PROGRAM POU
VAR
	
	i : INT := 0;
	f : REAL := 0.0;
	elapsed : TIME := TIME#0M0S0MS;
	today : DATE := DATE#2020-01-01;
	message : STRING := '';
	count : BYTE := 0;
	
	A AT %I* : BOOL := FALSE;
	B AT %I* : BOOL := FALSE;
	C AT %I* : BOOL := FALSE;
	D AT %Q* : BOOL := FALSE;
		
	op1 : INT := 1;
	op2 : INT := 2;
	res : REAL := 0.0;
	test : BOOL := FALSE;
	
	tmr1 : TON;
	
END_VAR

// Single line comment

(* 
	Multiple line comment
*)

// Structured Text statments

i := 0;
f := 0.0;
elapsed := T#1S;
today := D#2020-05-18;
message := 'Good Morning!';

// Operators (strongest to weakest binding)

res := MAX(op1,op2); // MAX() function

res := EXPT(op1, op2); // Exponentation operator

res := -op1; // Negation operator
B := NOT A; // NOT operator

res := op1 * op2; // * operator
res := op1 / op2; // / operator
res := op1 MOD op2; // MOD operator

res := op1 + op2; // + operator
res := op1 - op2; // - operator

test := op1 < op2; // < operator
test := op1 > op2; // > operator
test := op1 <= op2; // <= operator
test := op1 >= op2; // >= operator

test := op1 = op2; // = operator

C := A AND B; // AND operator

C := A XOR B; // XOR operator

C := A OR B; // OR operator

// IF statement

IF A = B THEN // IF statement
	D := TRUE;
END_IF

IF A = B THEN // IF-ELSE statement
	D := TRUE;
ELSE
	D := FALSE;
END_IF

IF A = B THEN // IF-ELSIF statement
	D := TRUE;
ELSIF A = C THEN
	D := FALSE;
END_IF

// CASE Statement

i := 0;

CASE i OF
	0: A := TRUE;
	1: B := TRUE;
	2: C := TRUE;
ELSE
	D := TRUE;
END_CASE

// FOR statement

f := 0.0;

FOR i := 0 TO 5 BY 1 DO // FOR loop
	f := f + i;
END_FOR

f := 0.0;

FOR i := 0 TO 5 BY 1 DO // FOR loop with EXIT statment
	f := f + i;
	
	IF f > 3 THEN
		EXIT;
	END_IF
END_FOR

// WHILE loop

i := 0;
f := 0.0;

WHILE f < 5 DO // WHILE loop
	f := f + i;
	i := i + 1;
END_WHILE

i := 0;
f := 0.0;

WHILE f < 5 DO // WHILE loop with EXIT statement
	f := f + i;
	i := i + 1;
	
	IF f > 3 THEN
		EXIT;
	END_IF
END_WHILE

// REPEAT loop

i := 0;
f := 0.0;

REPEAT // REPEAT loop
	f := f + i;
	i := i + 1;
UNTIL f >= 5
END_REPEAT

REPEAT // REPEAT loop with EXIT statment
	f := f + i;
	i := i + 1;
	
	IF f > 3 THEN
		EXIT;
	END_IF
UNTIL f = 5
END_REPEAT

// Timer

D := FALSE;
tmr1(IN := TRUE, PT := T#5S);

IF (tmr1.ET >= T#3S) THEN
	D := TRUE;
END_IF

END_PROGRAM

(* stored: Version 1.1.0.1, ProductVersion 3.1.4024.3
   POU POU: Id {3aa134d1-1501-444a-8c51-f815c03ebda5}, SpecialFunc None *)
